Staubli VAL3: Day5.dtx

string sInput
lists lResult
  [0]
    string sString
num nGrid[1 1]
lists lTemp
  [0]
    string sString
num nX1
num nY1
num nX2
num nY2
string sX1
string sY1
string sX2
string sY2
num nResRangeX
num nResRangeY
num nIntX
num nIntY
